FUNCTION_BLOCK HMI_EM_LogicExample EXTENDS FB_HMI_Base
VAR_INPUT
END_VAR
VAR_OUTPUT
END_VAR
VAR
	s_itfEmLogicExample1	: ITF_EM_LogicExample1; // Upgraded Interface from Control module
// Hmi Control Modules 
	s_hmiCmAxis1			: HMI_CM_Servo_Gain;
	s_hmiCmWaterInlet		: HMI_CM_Valve_Gain;
	s_hmiCmBelt				: HMI_CM_MotorDol_Gain;
	s_hmiCmHeightAdjuster	: HMI_CM_MotorDol_AF_Gain;
	
// Other
	s_fbLedRun				: FB_HmiLed;
	s_fbBtnStart			: FB_HmiButton;
END_VAR

SUPER^();

METHOD PUBLIC m_Main
SUPER^.m_Main();

// Upgrade the base-interface
IF NOT __QUERYINTERFACE(i_itfModule, s_itfEmLogicExample1) THEN
	RETURN;
END_IF

// Control modules
// Servo - Axis 1
s_hmiCmAxis1(
	i_itfModule		:= s_itfEmLogicExample1.p_itfCmAxis1, 
	i_eCfgMoveAbs	:= E_HMI_CM_SERVO_MoveAbsMode_Direction.MoveToModuloPosShortestWay);

// Valve - Valve 1
s_hmiCmWaterInlet(i_itfModule := s_itfEmLogicExample1.p_itfCmWaterInlet);

// MotorDOL - Belt motor
s_hmiCmBelt(i_itfModule := s_itfEmLogicExample1.p_itfCmBelt);

// Height adjuster motor
s_hmiCmHeightAdjuster(i_itfModule := s_itfEmLogicExample1.p_itfCmHeightAdjuster);
END_METHOD

END_FUNCTION_BLOCK

(* stored: Version 1.1.0.1, ProductVersion 3.1.4024.12
   POU HMI_EM_LogicExample: Id {61d96809-d0b2-4ef1-a07b-28187830b297}, SpecialFunc None
   Method m_Main: Id {3b79c43c-d8b5-470d-af6c-8adf9d16112d} *)
